INTERFACE I_EventEmitter EXTENDS __SYSTEM.IQueryInterface

METHOD PUBLIC OffEvent
VAR_INPUT
	EventName : T_MaxString;
	EventHandler : I_EventHandler;
END_VAR
END_METHOD

METHOD PUBLIC OnceEvent
VAR_INPUT
	EventName : T_MaxString;
	EventHandler : I_EventHandler;
END_VAR
END_METHOD

METHOD PUBLIC OnEvent
VAR_INPUT
	EventName : T_MaxString;
	EventHandler : I_EventHandler;
END_VAR
END_METHOD

END_INTERFACE

(* stored: Version 1.1.0.1, ProductVersion 3.1.4024.12
   Itf I_EventEmitter: Id {c55f25fc-a4d5-47c7-8a12-0023ae60d758}
   Method OffEvent: Id {cc0bcb0d-5cfc-48cb-adfb-7d9cc53f386b}
   Method OnceEvent: Id {fa95f361-7d3a-00a0-1a77-01b9b1274a14}
   Method OnEvent: Id {2e03d535-13cf-4113-b076-7f6e39ef2987} *)
